// SIMATIC S7-200 project (STEP 7-Micro/WIN), CPU 222 REL 01.00

ORGANIZATION_BLOCK MAIN:OB1
TITLE=【恒压供水控制系统（二）】
// 我实现了四个不同的恒压供水控制系统，这是第二个。
// 涉及多台水泵、变频器、压力传感器、自动/手动切换按钮、系统报警指示灯、水泵故障指示灯、系统运行指示灯和PID运行指示灯。
// 系统支持通过自动/手动切换按钮选择运行模式。在自动模式下，压力设定值固定为0.9 bar，系统通过 PID 控制器调节压力，根据当前压力值与设定值的偏差，计算 PID 输出值调整变频器运行。系统启动时，PID 启用标志置位，启用 PID 控制。系统根据压力情况动态调整水泵数量，例如，当压力低于阈值时，系统增加水泵数量；当压力高于阈值时，系统减少水泵数量。同时通过目标水泵数量和当前运行水泵编号动态控制水泵数量，且目标水泵数量始终保持在0到3之间，以避免系统尝试启动不存在的水泵，确保逻辑合理性。
// 水泵的启停过程有序进行，启动时由水泵启动延时定时器计时，确保切换平稳。例如，启动水泵1时，水泵1启动信号置位，同时水泵1运行指示灯点亮，且两者的状态始终互斥，避免出现启动信号为1而运行指示灯为0的冲突情况。系统避免频繁启停水泵，保护设备寿命。系统状态通过指示灯显示，变频器状态通过指示灯显示。
// 在手动模式下，压力设定值不同，操作员可通过水泵1手动启动按钮、水泵2手动启动按钮和水泵3手动启动按钮直接控制水泵。手动模式下有指示灯提示，手动操作设计安全。
// 系统有故障保护。当压力传感器故障输入为1时，表明传感器失效，此时 PID 启用标志立即置0，停止 PID 控制，防止压力失控，同时传感器故障时报警。水泵故障时有指示，可通过停止按钮中断运行，确保系统安全。
// 
// 
BEGIN
Network 1 // 网络标题
// 网络注释
LD     SM0.1
CALL   SBR_0:SBR0
Network 2
LD     I0.0
MOVR   0.9, VD104
NOT
MOVR   0.7, VD104
Network 3
LD     SM0.1
O      M0.0
INCB   VB300
Network 4
LD     I0.0
AD>=   VD250, VD212
AN     M0.1
LDN    I0.0
AD>=   VD250, VD208
OLD
TON    T37, +50
Network 5
LD     T37
AB<=   VB301, 1
EU
=      M0.1
INCB   VB301
Network 6
LDD<=  VD250, +1800
AN     M0.2
TON    T38, +100
Network 7
LD     T38
AB>    VB301, 0
EU
=      M0.2
DECB   VB301
Network 8
LD     M0.1
O      M0.3
S      M2.0, 1
Network 9
LD     M2.0
TON    T33, +1
=      Q1.5
Network 10
LD     T33
EU
=      M0.4
Network 11
LD     M0.4
S      M2.1, 1
INCB   VB300
Network 12
LD     M2.1
TON    T34, +2
Network 13
LD     T34
EU
=      M0.5
R      M2.1, 1
Network 14
LD     M0.5
S      M2.2, 1
Network 15
LD     M2.2
TON    T39, +30
Network 16
LD     T39
EU
=      M0.6
R      M2.2, 1
R      M2.0, 1
Network 17
LDB>   VB300, 3
MOVB   1, VB300
Network 18
LDB=   VB301, 0
A      SM0.4
EU
INVD   VD310
Network 19
LDD>=  VD310, +180
EU
=      M0.3
MOVD   +0, VD310
Network 20
LDB<>  VB301, 0
MOVD   +0, VD310
Network 21
LD     SM0.1
O      M0.0
O      M0.6
AB=    VB300, 1
O      Q0.1
AN     M0.3
AN     M0.4
AN     Q0.0
=      Q0.1
Network 22
LD     M0.6
AB=    VB300, 2
O      Q0.3
AN     M0.3
AN     M0.4
AN     Q0.2
=      Q0.3
Network 23
LD     M0.6
AB=    VB300, 3
O      Q0.5
AN     M0.3
AN     M0.4
AN     Q0.4
=      Q0.5
Network 24
LD     M0.5
O      Q0.0
LDB=   VB300, 2
AB>    VB301, 0
LDB=   VB300, 3
AB>    VB301, 1
OLD
ALD
AN     Q0.1
=      Q0.0
Network 25
LD     M0.5
O      Q0.2
LDB=   VB300, 3
AB>    VB301, 0
LDB=   VB300, 1
AB>    VB301, 1
OLD
ALD
AN     Q0.3
=      Q0.2
Network 26
LD     M0.5
O      Q0.4
LDB=   VB300, 1
AB>    VB301, 0
LDB=   VB300, 2
AB>    VB301, 1
OLD
ALD
AN     Q0.5
=      Q0.4
Network 27
LD     I0.0
=      Q1.0
Network 28
LDN    I0.1
O      M3.1
A      I0.2
=      M3.1
Network 29
LD     SM0.5
O      M3.2
A      M3.1
O      I0.5
=      Q1.1
Network 30
LD     SM0.5
O      M3.3
A      I0.3
O      I0.5
=      Q1.2
Network 31
LD     SM0.5
O      M3.4
A      I0.0
O      I0.5
=      Q1.3
Network 32
LD     I0.4
O      M3.2
A      M3.1
=      M3.2
Network 33
LD     I0.4
O      M3.3
A      I0.3
=      M3.3
Network 34
LD     I0.4
O      M3.4
A      I0.0
=      M3.4
Network 35
LD     M3.1
AN     M3.2
LD     I0.3
AN     M3.3
OLD
LD     I0.0
AN     M3.4
OLD
O      I0.5
=      Q1.4
Network 36
LD     M3.1
O      I0.3
=      M3.0
MOVB   0, VB300
MOVB   0, VB301
ED
=      M0.0
END_ORGANIZATION_BLOCK

SUBROUTINE_BLOCK SBR_0:SBR0
TITLE=子例行程序注释
BEGIN
Network 1 // 网络标题
// 网络注释
LD     SM0.0
MOVD   +1800, VD204
MOVD   +22400, VD208
MOVD   +28800, VD212
MOVR   0.25, VD112
MOVR   0.2, VD116
MOVR   30.0, VD120
MOVR   0.0, VD124
MOVB   200, SMB34
ATCH   INT_0:INT0, 10
END_SUBROUTINE_BLOCK

INTERRUPT_BLOCK INT_0:INT0
TITLE=中断例行程序注释
BEGIN
Network 1 // 网络标题
// 网络注释
LD     SM0.0
ITD    AIW0, AC0
DTR    AC0, AC0
/R     32000.0, AC0
PID    VB100, 0
MOVR   VD108, AC0
MOVR   VD108, AC0
*R     32000.0, AC0
Network 2
LDR<=  AC0, VD204
OW>    T39, +25
MOVD   VD204, AC0
Network 3
LD     SM0.0
ROUND  AC0, AC0
MOVD   AC0, VD250
DTI    AC0, AC0
MOVW   AC0, AQW0
END_INTERRUPT_BLOCK
